// TIA Portal V17 export
// export: Created 2023-03-06T02:05:26.0452917Z, ExportSetting WithDefaults, DisplayName Totally Integrated Automation Portal, DisplayVersion V17 Update 4, DisplayName TIA Portal Openness, DisplayVersion V17 Update 4, DisplayName TIA Portal Version Control Interface, DisplayVersion V17, DisplayName STEP 7 Professional, DisplayVersion V17 Update 4, DisplayName STEP 7 Safety, DisplayVersion V17, DisplayName WinCC Professional, DisplayVersion V17 Update 4
TYPE "BMS_BB"
// stored: IsFailsafeCompliant false
   STRUCT
      iHeartBeatCount : Int;   // Heartbeat
      wCmd : Word;   // Command
      wFltClearCmd : Word;   // Fault_Clear
      iHeartBeatFb : Int;   // Heartbeat
      wPwrOnHvSt : Word;   // PowerOn
      wSMstatusSt : Word;   // Status
      iNBRconnectCount : Int;   // Number_HV_Connected
      rEnergyAvlChaMeas : Real;   // System_Remain_Ch_Energy
      rEnergyAvlDschMeas : Real;   // System_Remain_Dh_Energy
      wWarn1 : Word;   // Warning_1
      wWarn2 : Word;   // Warning_2
      wWarn3 : Word;   // Warning_3
      wWarn4 : Word;   // Warning_4
      xInitSt : Bool;   // Word Status = 0
      xNormOpSt : Bool;   // Word Status = 1
      xFullChaSt : Bool;   // Word Status = 2
      xFullDschSt : Bool;   // Word Status = 3
      xWarnSt : Bool;   // Word Status = 4
      xFltSt : Bool;   // Word Status = 5
      rVdcMeas : Real;   // Voltage
      rIdcMeas : Real;   // Current
      rSOCmeas : Real;   // SOC
      rSOHmeas : Real;   // SOH
      rVcellMaxMeas : Real;   // Max_Cell_Volt
      rVcellMinMeas : Real;   // Min_Cell_Volt
      rVcellAvgMeas : Real;   // Avg_Cell_Volt
      iTcellMaxMeas : Int;   // Max_Cell_Temp
      iTcellMinMeas : Int;   // Min_Cell_Temp
      iTcellAvgMeas : Int;   // Avg_Cell_Temp
      rIchaLim : Real;   // Max_Charge_Curr
      rIdschLim : Real;   // Max_Discharge_Curr
      iNBRtotalCount { S7_SetPoint := 'True'} : Int;   // Total Number of Rack
   END_STRUCT;
END_TYPE
